FUNCTION_BLOCK E_N_TABLE (* Generation of a finite train of separate events,table driven *)
  (* Standard: 61499-1; Classification: Event processing; Function: Event train generation *)
  (* Version 0.1, 2002-01-29, JHC, Rockwell Automation, XML version *)
  (* Version 0.0, 1998-04-10, JHC, Rockwell Automation, SRC version *)
  (* Compiler header: package fb.rt.events; *)
  (* Compiler Java IBM VisualAge 3.0 *)
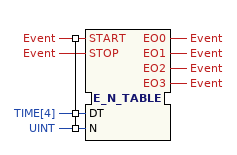
  EVENT_INPUT
    START WITH DT, N;
    STOP;
  END_EVENT
  EVENT_OUTPUT
    EO0; (* N events at periods DT,starting at DT[0]after EI *)
    EO1;
    EO2;
    EO3; (* Maximum number of events=DT array size *)
  END_EVENT
  VAR_INPUT
    DT : ARRAY [0..3] OF TIME; (* Periods between events,maximum is implementation dependent *)
    N : UINT; (* Number of events to generate,up to size of DT *)
  END_VAR
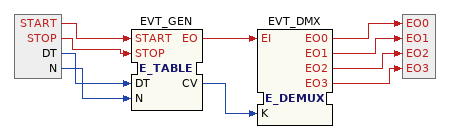
  FBS
    EVT_GEN : E_TABLE;
    EVT_DMX : E_DEMUX;
  END_FBS
  EVENT_CONNECTIONS
    START TO EVT_GEN.START;
    STOP TO EVT_GEN.STOP;
    EVT_GEN.EO TO EVT_DMX.EI;
    EVT_DMX.EO0 TO EO0;
    EVT_DMX.EO1 TO EO1;
    EVT_DMX.EO2 TO EO2;
    EVT_DMX.EO3 TO EO3;
  END_CONNECTIONS
  DATA_CONNECTIONS
    DT TO EVT_GEN.DT;
    N TO EVT_GEN.N;
    EVT_GEN.CV TO EVT_DMX.K;
  END_CONNECTIONS
END_FUNCTION_BLOCK
